{attribute 'qualified_only'}
VAR_GLOBAL
	{attribute 'federico' := 'The best'}
	Body : ARRAY [1..10] OF STRING;
	test : json;
END_VAR

(* stored: Version 1.1.0.1, ProductVersion 3.1.4022.12
   GVL GVL: Id {d51db366-947e-48a2-9a01-f59b16646812} *)
